// FB_ListRecipeFiles: Scans the recipe folder and fills GVL_Recipe.aAvailableFiles with metadata from JSON files
FUNCTION_BLOCK FB_ListRecipeFiles
VAR_INPUT
	bExecute : BOOL; // Start the file listing process
END_VAR
VAR_OUTPUT
	bBusy       : BOOL; // Indicates the block is busy
    bError      : BOOL; // Indicates an error occurred
    nErrId      : UDINT; // Error code if any
	bDone   	: BOOL;

END_VAR
VAR
	fbEnumFiles     : FB_EnumFindFileList;
    fbFileTime      : FB_FileTime64ToTzSpecificLocalTime;
    fbHeaderHandler : FB_RecipeHeaderHandler;

    aFindBuffer     : ARRAY[0..49] OF ST_FindFileEntry;
    nFoundFiles     : UDINT;
    iFileIndex      : INT;
    iStep           : INT;
    bExecutePrev    : BOOL;
    bStart          : BOOL;
    bHeaderHandlerReset : BOOL;
    bHeaderHandlerExecute : BOOL;
END_VAR

bStart := NOT bExecutePrev AND bExecute;
bExecutePrev := bExecute;

CASE iStep OF

0:
    IF bStart THEN
        bBusy := TRUE;
        bDone := FALSE;
        bError := FALSE;
        nErrId := 0;
        iFileIndex := 0;
        bHeaderHandlerReset := FALSE;
        bHeaderHandlerExecute := FALSE;

        fbEnumFiles(
            sNetId := '',
            sPathName := 'C:/TwinCAT/Recipes/*.json',
            eCmd := eEnumCmd_First,
            pFindList := ADR(aFindBuffer),
            cbFindList := SIZEOF(aFindBuffer),
            bExecute := TRUE
        );

        iStep := 10;
    END_IF

10:
    fbEnumFiles(bExecute := FALSE);
    IF NOT fbEnumFiles.bBusy THEN
        IF fbEnumFiles.bError THEN
            bError := TRUE;
            nErrId := fbEnumFiles.nErrId;
            iStep := 100;
        ELSE
            nFoundFiles := fbEnumFiles.nFindFiles;
            IF nFoundFiles > 0 THEN
                iStep := 20;
            ELSE
                bDone := TRUE;
                iStep := 100;
            END_IF
        END_IF
    END_IF

20:
    IF iFileIndex < TO_INT(nFoundFiles) AND iFileIndex <= 49 THEN
        IF NOT fbHeaderHandler.bBusy THEN
            IF bHeaderHandlerReset THEN
                // Wait one cycle with bExecute := FALSE
                fbHeaderHandler(bExecute := FALSE);
                bHeaderHandlerReset := FALSE;
                iStep := 25;
            ELSIF NOT bHeaderHandlerExecute THEN
                // Fill file name and timestamp
                GVL_Recipe.aAvailableFiles[iFileIndex].sFileName := aFindBuffer[iFileIndex].sFileName;
                fbFileTime(
                    in := FILETIME_TO_FILETIME64(aFindBuffer[iFileIndex].lastWriteTime),
                    tzInfo := WEST_EUROPE_TZI
                );
                GVL_Recipe.aAvailableFiles[iFileIndex].dtLastModified := FILETIME64_TO_DT(fbFileTime.out);

                // Trigger header parser
                fbHeaderHandler(
                    sFileName := CONCAT('C:/TwinCAT/Recipes/', aFindBuffer[iFileIndex].sFileName),
                    iTargetIndex := iFileIndex,
                    bExecute := TRUE
                );
                bHeaderHandlerExecute := fbHeaderHandler.bDone;
            ELSE
				
                iStep := 30;
				
            END_IF
        END_IF
    ELSE
        bDone := TRUE;
        iStep := 100;
    END_IF

25:
    fbHeaderHandler(bExecute := FALSE);
    iStep := 20;

30:
    fbHeaderHandler(bExecute := FALSE);
    IF NOT fbHeaderHandler.bBusy THEN
        IF fbHeaderHandler.bError THEN
            bError := TRUE;
            nErrId := fbHeaderHandler.nErrId;
            iStep := 100;
        ELSIF fbHeaderHandler.bDone THEN
            bHeaderHandlerReset := TRUE;
            bHeaderHandlerExecute := FALSE;
            iFileIndex := iFileIndex + 1;
            iStep := 20;
        END_IF
    END_IF

100:
    bBusy := FALSE;
    IF NOT bExecute THEN
        iStep := 0;
    END_IF
END_CASE

END_FUNCTION_BLOCK

(* stored: Version 1.1.0.1, ProductVersion 3.1.4024.12
   POU FB_ListRecipeFiles: Id {c0094d53-68e1-453f-9c4e-bed934c9b18b}, SpecialFunc None *)
